Staubli VAL3: IOInterface.pjx

Parameters version=s7.7.2 stackSize=5000 millimeterUnit=true
Program file=init.pgx
Program file=readAll.pgx
Program file=start.pgx
Program file=stop.pgx
Program file=writeSingle.pgx
Data file=IOInterface.dtx
Library alias=IOModule path=Disk://ros_libs/IOModule/IOModule.pjx autoload=true password=
